% RSLogix 500 project I2P-JOB21-ADAM BOCZKIEWICZ_BAK047.RSS, saved by version 10.00.00.00 %
PROJECT "ML04A"    % processor: Bul.1763 MicroLogix 1100 Series B %

PROGRAM FILES
  LAD 2   5 rungs

DATA FILES
  O0 OUTPUT  4 elements
  I1 INPUT  6 elements
  S2 STATUS  66 elements
  B3 BINARY  1 elements
  T4 TIMER  1 elements
  C5 COUNTER  1 elements
  R6 CONTROL  1 elements
  N7 INTEGER  1 elements
  F8 FLOAT  1 elements

LADDER 2
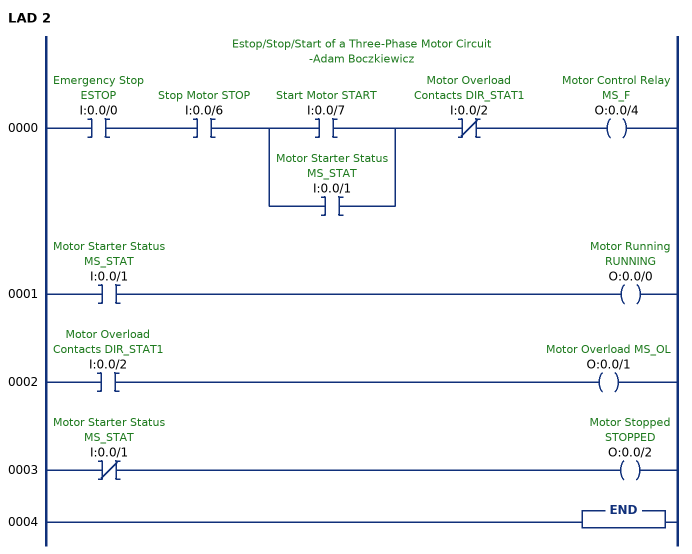
% Rung: 0 %
% Estop/Stop/Start of a Three-Phase Motor Circuit
% -Adam Boczkiewicz %
SOR XIC I:0.0/0 XIC I:0.0/6 BST XIC I:0.0/7 NXB XIC I:0.0/1 BND XIO I:0.0/2 OTE O:0.0/4 EOR
%   I:0.0/0  ESTOP  "Emergency Stop" %
%   I:0.0/6  STOP  "Stop Motor" %
%   I:0.0/7  START  "Start Motor" %
%   I:0.0/1  MS_STAT  "Motor Starter Status" %
%   I:0.0/2  DIR_STAT1  "Motor Overload Contacts" %
%   O:0.0/4  MS_F  "Motor Control Relay" %
% Rung: 1 %
SOR XIC I:0.0/1 OTE O:0.0/0 EOR
%   I:0.0/1  MS_STAT  "Motor Starter Status" %
%   O:0.0/0  RUNNING  "Motor Running" %
% Rung: 2 %
SOR XIC I:0.0/2 OTE O:0.0/1 EOR
%   I:0.0/2  DIR_STAT1  "Motor Overload Contacts" %
%   O:0.0/1  MS_OL  "Motor Overload" %
% Rung: 3 %
SOR XIO I:0.0/1 OTE O:0.0/2 EOR
%   I:0.0/1  MS_STAT  "Motor Starter Status" %
%   O:0.0/2  STOPPED  "Motor Stopped" %
% Rung: 4 %
SOR END EOR

OTHER DOCUMENTED ADDRESSES
  B3:0/0  JBF  "Jog Bit FWD"
  B3:0/1  JBR  "Jog Bit Reverse"
  B3:0/2  FB  "Foward Bit"
  B3:0/3  RB  "Reverse Bit"
  B3:0/4  DCF  "Last Direction Foward Bit"
  B3:0/5  DCR  "Last Direction Reverse Bit"
  B3:0/6  YB  "Yellow Bit"
  I:0.0/3  ON_MODE  "Mode: On Position"
  I:0.0/4  AUTO_MODE  "Mode: Auto Postion"
  I:0.0/5  RUN_JO  "Run/Jog Mode"
  I:0.0/8  REV  "Jog Motor"
  I:0.0/9  LO_LVL  "Low Level Switch"
  JOG  
  MO  
  O:0.0/3  FULL  "Tank Full"
  O:0.0/5  CR2  "Valve Control"
  T4:0/TT  TT

COMMENTS NOT ATTACHED TO A CURRENT RUNG
  B3:0/0: Fwd-Rev-Jog Using two position selector switches for a 1P motor
    Adam Boczkiewicz

DATA TABLE (non-zero values as saved)
DATA T4
% .PRE .ACC %
% T4:0 % 8 0
DATA C5
% .PRE .ACC %
% C5:0 % 16 1
